PROGRAM Automatic_POU
VAR
	nStep 			:INT;
	bHlatMode,bNextStep		:BOOL;
END_VAR

//實例化

CASE  nStep OF
	0:
		M_Openbox1.Process(bHlatMode);
		M_Sealing2.Process(FALSE);
		M_LoadPic3.Process(FALSE);
		M_UnloadNG4.Process(FALSE);
		M_DualServo.Process(FALSE);
		M_StackComv5.Process(FALSE);
		M_RBStack6.Process(FALSE);
END_CASE
IF bNextStep THEN
	M_Openbox1.HaltStepContiune();
	bNextStep:=FALSE;
END_IF

END_PROGRAM

(* stored: Version 1.1.0.1, ProductVersion 3.1.4024.16
   POU Automatic_POU: Id {d539cfdc-f8c2-4c03-ad90-2b9ea190d71a}, SpecialFunc None *)
